Staubli VAL3: main.pgx

public program main()
begin
end
